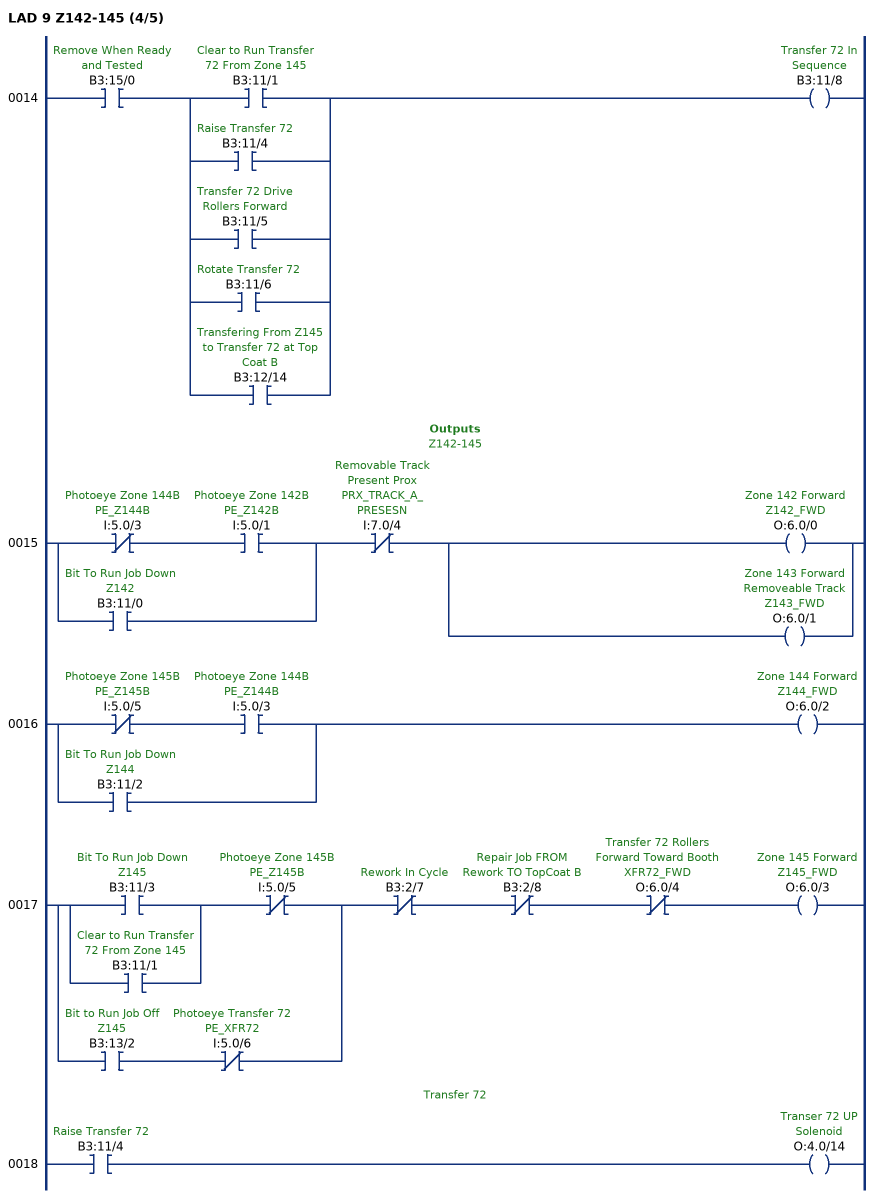
% Rung: 14 %
SOR XIC B3:15/0 BST XIC B3:11/1 NXB XIC B3:11/4 NXB XIC B3:11/5 NXB XIC B3:11/6 NXB XIC B3:12/14 BND OTE B3:11/8 EOR
%   B3:15/0  "Remove When Ready and Tested" %
%   B3:11/1  "Clear to Run Transfer 72 From Zone 145" %
%   B3:11/4  "Raise Transfer 72" %
%   B3:11/5  "Transfer 72 Drive Rollers Forward" %
%   B3:11/6  "Rotate Transfer 72" %
%   B3:12/14  "Transfering From Z145 to Transfer 72 at Top Coat B" %
%   B3:11/8  "Transfer 72 In Sequence" %
% Rung: 15 %
% TITLE: Outputs %
% Z142-145 %
SOR BST XIO I:5.0/3 XIC I:5.0/1 NXB XIC B3:11/0 BND XIO I:7.0/4 BST OTE O:6.0/0 NXB OTE O:6.0/1 BND EOR
%   I:5.0/3  PE_Z144B  "Photoeye Zone 144B" %
%   I:5.0/1  PE_Z142B  "Photoeye Zone 142B" %
%   B3:11/0  "Bit To Run Job Down Z142" %
%   I:7.0/4  PRX_TRACK_A_PRESESN  "Removable Track Present Prox" %
%   O:6.0/0  Z142_FWD  "Zone 142 Forward" %
%   O:6.0/1  Z143_FWD  "Zone 143 Forward Removeable Track" %
% Rung: 16 %
SOR BST XIO I:5.0/5 XIC I:5.0/3 NXB XIC B3:11/2 BND OTE O:6.0/2 EOR
%   I:5.0/5  PE_Z145B  "Photoeye Zone 145B" %
%   I:5.0/3  PE_Z144B  "Photoeye Zone 144B" %
%   B3:11/2  "Bit To Run Job Down Z144" %
%   O:6.0/2  Z144_FWD  "Zone 144 Forward" %
% Rung: 17 %
SOR BST BST XIC B3:11/3 NXB XIC B3:11/1 BND XIO I:5.0/5 NXB XIC B3:13/2 XIO I:5.0/6 BND XIO B3:2/7 XIO B3:2/8 XIO O:6.0/4 OTE O:6.0/3 EOR
%   B3:11/3  "Bit To Run Job Down Z145" %
%   B3:11/1  "Clear to Run Transfer 72 From Zone 145" %
%   I:5.0/5  PE_Z145B  "Photoeye Zone 145B" %
%   B3:13/2  "Bit to Run Job Off Z145" %
%   I:5.0/6  PE_XFR72  "Photoeye Transfer 72" %
%   B3:2/7  "Rework In Cycle" %
%   B3:2/8  "Repair Job FROM Rework TO TopCoat B" %
%   O:6.0/4  XFR72_FWD  "Transfer 72 Rollers Forward Toward Booth" %
%   O:6.0/3  Z145_FWD  "Zone 145 Forward" %
% Rung: 18 %
% Transfer 72 %
SOR XIC B3:11/4 OTE O:4.0/14 EOR
%   B3:11/4  "Raise Transfer 72" %
%   O:4.0/14  "Transer 72 UP Solenoid" %

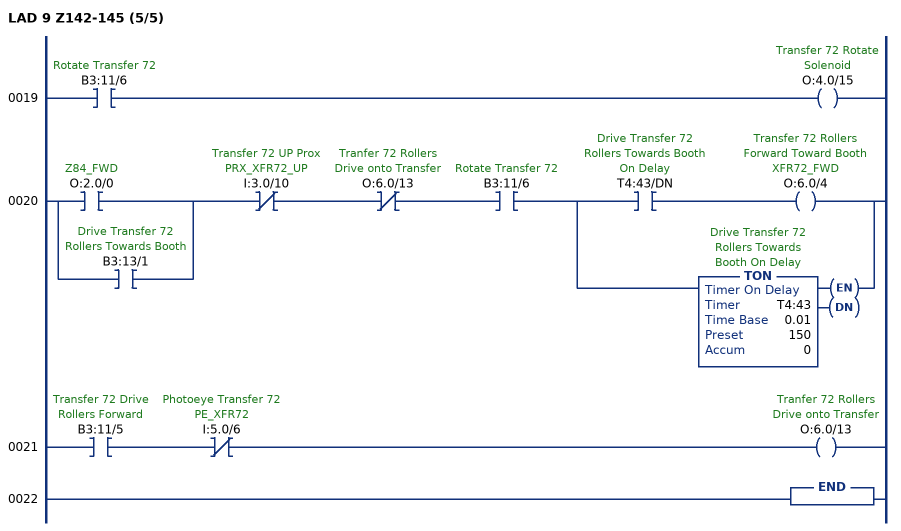
% Rung: 19 %
SOR XIC B3:11/6 OTE O:4.0/15 EOR
%   B3:11/6  "Rotate Transfer 72" %
%   O:4.0/15  "Transfer 72 Rotate Solenoid" %
% Rung: 20 %
SOR BST XIC O:2.0/0 NXB XIC B3:13/1 BND XIO I:3.0/10 XIO O:6.0/13 XIC B3:11/6 BST XIC T4:43/DN OTE O:6.0/4 NXB TON T4:43 0.01 150 0 BND EOR
%   O:2.0/0  Z84_FWD %
%   B3:13/1  "Drive Transfer 72 Rollers Towards Booth" %
%   I:3.0/10  PRX_XFR72_UP  "Transfer 72 UP Prox" %
%   O:6.0/13  "Tranfer 72 Rollers Drive onto Transfer" %
%   B3:11/6  "Rotate Transfer 72" %
%   T4:43  "Drive Transfer 72 Rollers Towards Booth On Delay" %
%   O:6.0/4  XFR72_FWD  "Transfer 72 Rollers Forward Toward Booth" %
% Rung: 21 %
SOR XIC B3:11/5 XIO I:5.0/6 OTE O:6.0/13 EOR
%   B3:11/5  "Transfer 72 Drive Rollers Forward" %
%   I:5.0/6  PE_XFR72  "Photoeye Transfer 72" %
%   O:6.0/13  "Tranfer 72 Rollers Drive onto Transfer" %
% Rung: 22 %
SOR END EOR

LADDER 10 "TO_GLAZE"
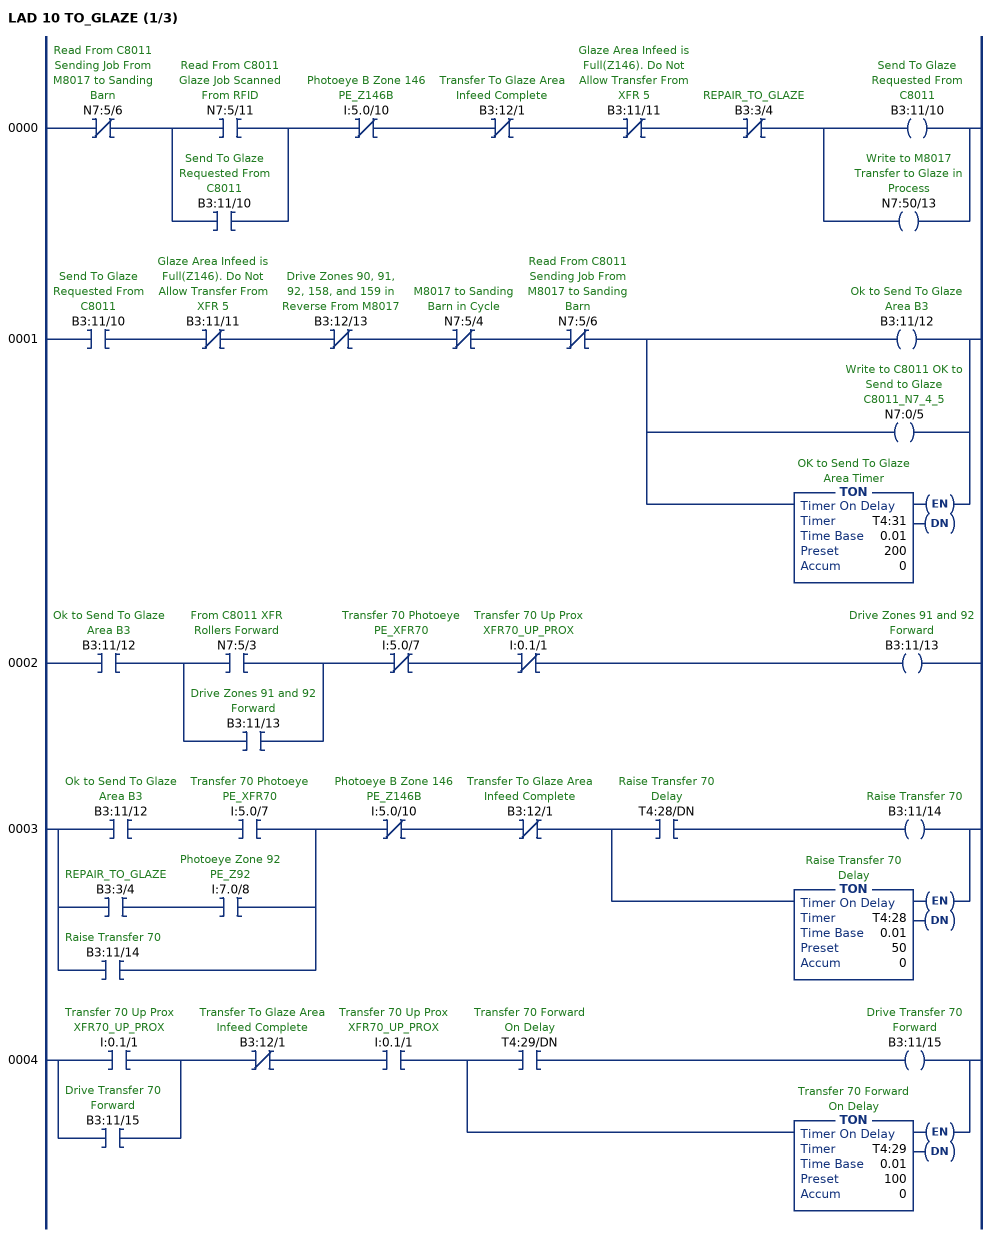
% Rung: 0 %
SOR XIO N7:5/6 BST XIC N7:5/11 NXB XIC B3:11/10 BND XIO I:5.0/10 XIO B3:12/1 XIO B3:11/11 XIO B3:3/4 BST OTE B3:11/10 NXB OTE N7:50/13 BND EOR
%   N7:5/6  "Read From C8011 Sending Job From M8017 to Sanding Barn" %
%   N7:5/11  "Read From C8011 Glaze Job Scanned From RFID" %
%   B3:11/10  "Send To Glaze Requested From C8011" %
%   I:5.0/10  PE_Z146B  "Photoeye B Zone 146" %
%   B3:12/1  "Transfer To Glaze Area Infeed Complete" %
%   B3:11/11  "Glaze Area Infeed is Full(Z146). Do Not Allow Transfer From XFR 5" %
%   B3:3/4  REPAIR_TO_GLAZE %
%   N7:50/13  "Write to M8017 Transfer to Glaze in Process" %
% Rung: 1 %
SOR XIC B3:11/10 XIO B3:11/11 XIO B3:12/13 XIO N7:5/4 XIO N7:5/6 BST BST OTE B3:11/12 NXB OTE N7:0/5 BND NXB TON T4:31 0.01 200 0 BND EOR
%   B3:11/10  "Send To Glaze Requested From C8011" %
%   B3:11/11  "Glaze Area Infeed is Full(Z146). Do Not Allow Transfer From XFR 5" %
%   B3:12/13  "Drive Zones 90, 91, 92, 158, and 159 in Reverse From M8017" %
%   N7:5/4  "M8017 to Sanding Barn in Cycle" %
%   N7:5/6  "Read From C8011 Sending Job From M8017 to Sanding Barn" %
%   B3:11/12  B3  "Ok to Send To Glaze Area" %
%   N7:0/5  C8011_N7_4_5  "Write to C8011 OK to Send to Glaze" %
%   T4:31  "OK to Send To Glaze Area Timer" %
% Rung: 2 %
SOR XIC B3:11/12 BST XIC N7:5/3 NXB XIC B3:11/13 BND XIO I:5.0/7 XIO I:0.1/1 OTE B3:11/13 EOR
%   B3:11/12  B3  "Ok to Send To Glaze Area" %
%   N7:5/3  "From C8011 XFR Rollers Forward" %
%   B3:11/13  "Drive Zones 91 and 92 Forward" %
%   I:5.0/7  PE_XFR70  "Transfer 70 Photoeye" %
%   I:0.1/1  XFR70_UP_PROX  "Transfer 70 Up Prox" %
% Rung: 3 %
SOR BST XIC B3:11/12 XIC I:5.0/7 NXB XIC B3:3/4 XIC I:7.0/8 NXB XIC B3:11/14 BND XIO I:5.0/10 XIO B3:12/1 BST XIC T4:28/DN OTE B3:11/14 NXB TON T4:28 0.01 50 0 BND EOR
%   B3:11/12  B3  "Ok to Send To Glaze Area" %
%   I:5.0/7  PE_XFR70  "Transfer 70 Photoeye" %
%   B3:3/4  REPAIR_TO_GLAZE %
%   I:7.0/8  PE_Z92  "Photoeye Zone 92" %
%   B3:11/14  "Raise Transfer 70" %
%   I:5.0/10  PE_Z146B  "Photoeye B Zone 146" %
%   B3:12/1  "Transfer To Glaze Area Infeed Complete" %
%   T4:28  "Raise Transfer 70 Delay" %
% Rung: 4 %
SOR BST XIC I:0.1/1 NXB XIC B3:11/15 BND XIO B3:12/1 XIC I:0.1/1 BST XIC T4:29/DN OTE B3:11/15 NXB TON T4:29 0.01 100 0 BND EOR
%   I:0.1/1  XFR70_UP_PROX  "Transfer 70 Up Prox" %
%   B3:11/15  "Drive Transfer 70 Forward" %
%   B3:12/1  "Transfer To Glaze Area Infeed Complete" %
%   T4:29  "Transfer 70 Forward On Delay" %

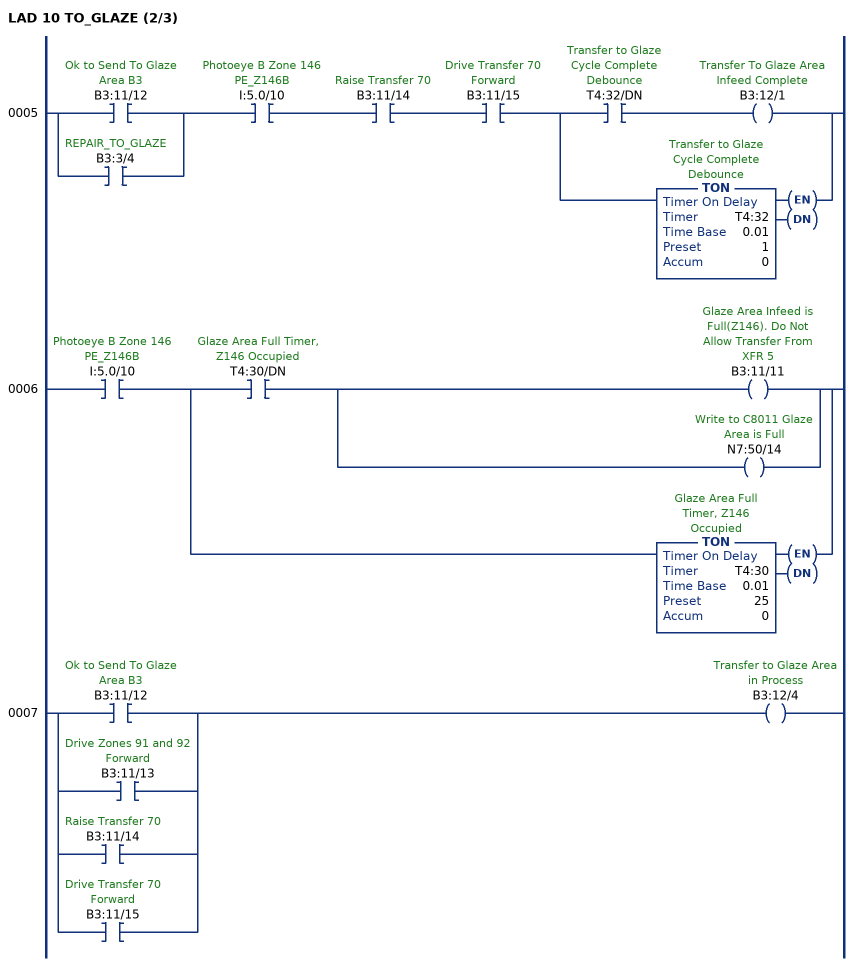
% Rung: 5 %
SOR BST XIC B3:11/12 NXB XIC B3:3/4 BND XIC I:5.0/10 XIC B3:11/14 XIC B3:11/15 BST XIC T4:32/DN OTE B3:12/1 NXB TON T4:32 0.01 1 0 BND EOR
%   B3:11/12  B3  "Ok to Send To Glaze Area" %
%   B3:3/4  REPAIR_TO_GLAZE %
%   I:5.0/10  PE_Z146B  "Photoeye B Zone 146" %
%   B3:11/14  "Raise Transfer 70" %
%   B3:11/15  "Drive Transfer 70 Forward" %
%   T4:32  "Transfer to Glaze Cycle Complete Debounce" %
%   B3:12/1  "Transfer To Glaze Area Infeed Complete" %
% Rung: 6 %
SOR XIC I:5.0/10 BST XIC T4:30/DN BST OTE B3:11/11 NXB OTE N7:50/14 BND NXB TON T4:30 0.01 25 0 BND EOR
%   I:5.0/10  PE_Z146B  "Photoeye B Zone 146" %
%   T4:30  "Glaze Area Full Timer, Z146 Occupied" %
%   B3:11/11  "Glaze Area Infeed is Full(Z146). Do Not Allow Transfer From XFR 5" %
%   N7:50/14  "Write to C8011 Glaze Area is Full" %
% Rung: 7 %
SOR BST XIC B3:11/12 NXB XIC B3:11/13 NXB XIC B3:11/14 NXB XIC B3:11/15 BND OTE B3:12/4 EOR
%   B3:11/12  B3  "Ok to Send To Glaze Area" %
%   B3:11/13  "Drive Zones 91 and 92 Forward" %
%   B3:11/14  "Raise Transfer 70" %
%   B3:11/15  "Drive Transfer 70 Forward" %
%   B3:12/4  "Transfer to Glaze Area in Process" %

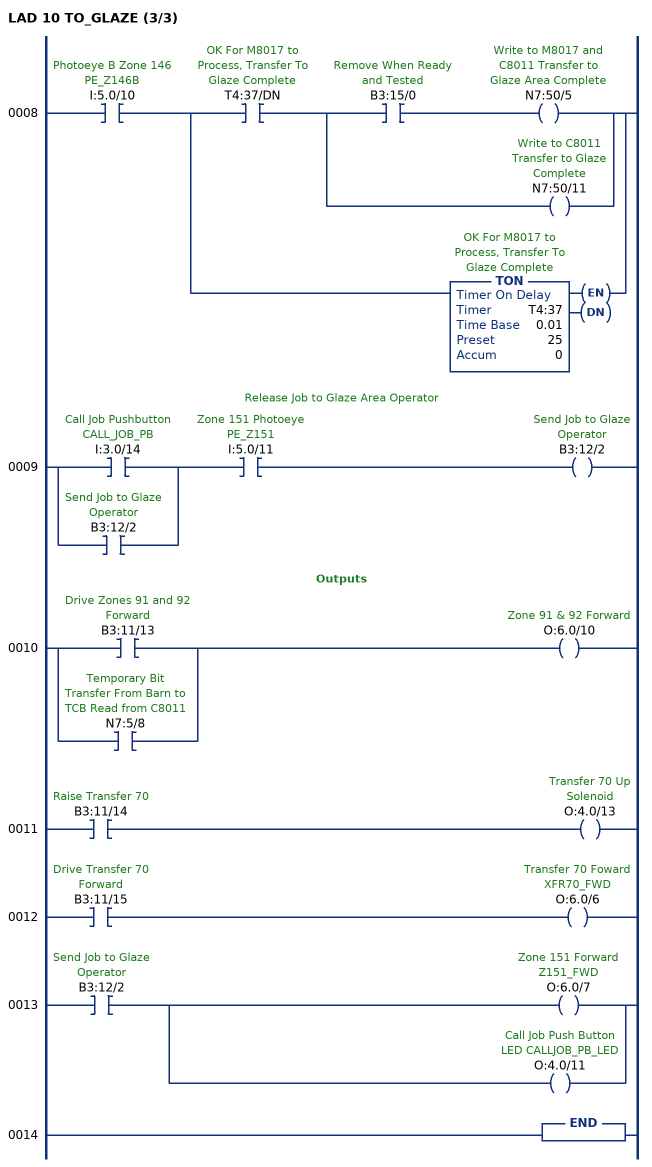
% Rung: 8 %
SOR XIC I:5.0/10 BST XIC T4:37/DN BST XIC B3:15/0 OTE N7:50/5 NXB OTE N7:50/11 BND NXB TON T4:37 0.01 25 0 BND EOR
%   I:5.0/10  PE_Z146B  "Photoeye B Zone 146" %
%   T4:37  "OK For M8017 to Process, Transfer To Glaze Complete" %
%   B3:15/0  "Remove When Ready and Tested" %
%   N7:50/5  "Write to M8017 and C8011 Transfer to Glaze Area Complete" %
%   N7:50/11  "Write to C8011 Transfer to Glaze Complete" %
% Rung: 9 %
% Release Job to Glaze Area Operator %
SOR BST XIC I:3.0/14 NXB XIC B3:12/2 BND XIC I:5.0/11 OTE B3:12/2 EOR
%   I:3.0/14  CALL_JOB_PB  "Call Job Pushbutton" %
%   B3:12/2  "Send Job to Glaze Operator" %
%   I:5.0/11  PE_Z151  "Zone 151 Photoeye" %
% Rung: 10 %
% TITLE: Outputs %
SOR BST XIC B3:11/13 NXB XIC N7:5/8 BND OTE O:6.0/10 EOR
%   B3:11/13  "Drive Zones 91 and 92 Forward" %
%   N7:5/8  "Temporary Bit Transfer From Barn to TCB Read from C8011" %
%   O:6.0/10  "Zone 91 & 92 Forward" %
% Rung: 11 %
SOR XIC B3:11/14 OTE O:4.0/13 EOR
%   B3:11/14  "Raise Transfer 70" %
%   O:4.0/13  "Transfer 70 Up Solenoid" %
% Rung: 12 %
SOR XIC B3:11/15 OTE O:6.0/6 EOR
%   B3:11/15  "Drive Transfer 70 Forward" %
%   O:6.0/6  XFR70_FWD  "Transfer 70 Foward" %
% Rung: 13 %
SOR XIC B3:12/2 BST OTE O:6.0/7 NXB OTE O:4.0/11 BND EOR
%   B3:12/2  "Send Job to Glaze Operator" %
%   O:6.0/7  Z151_FWD  "Zone 151 Forward" %
%   O:4.0/11  CALLJOB_PB_LED  "Call Job Push Button LED" %
% Rung: 14 %
SOR END EOR

LADDER 11 "FROM_GLAZE"
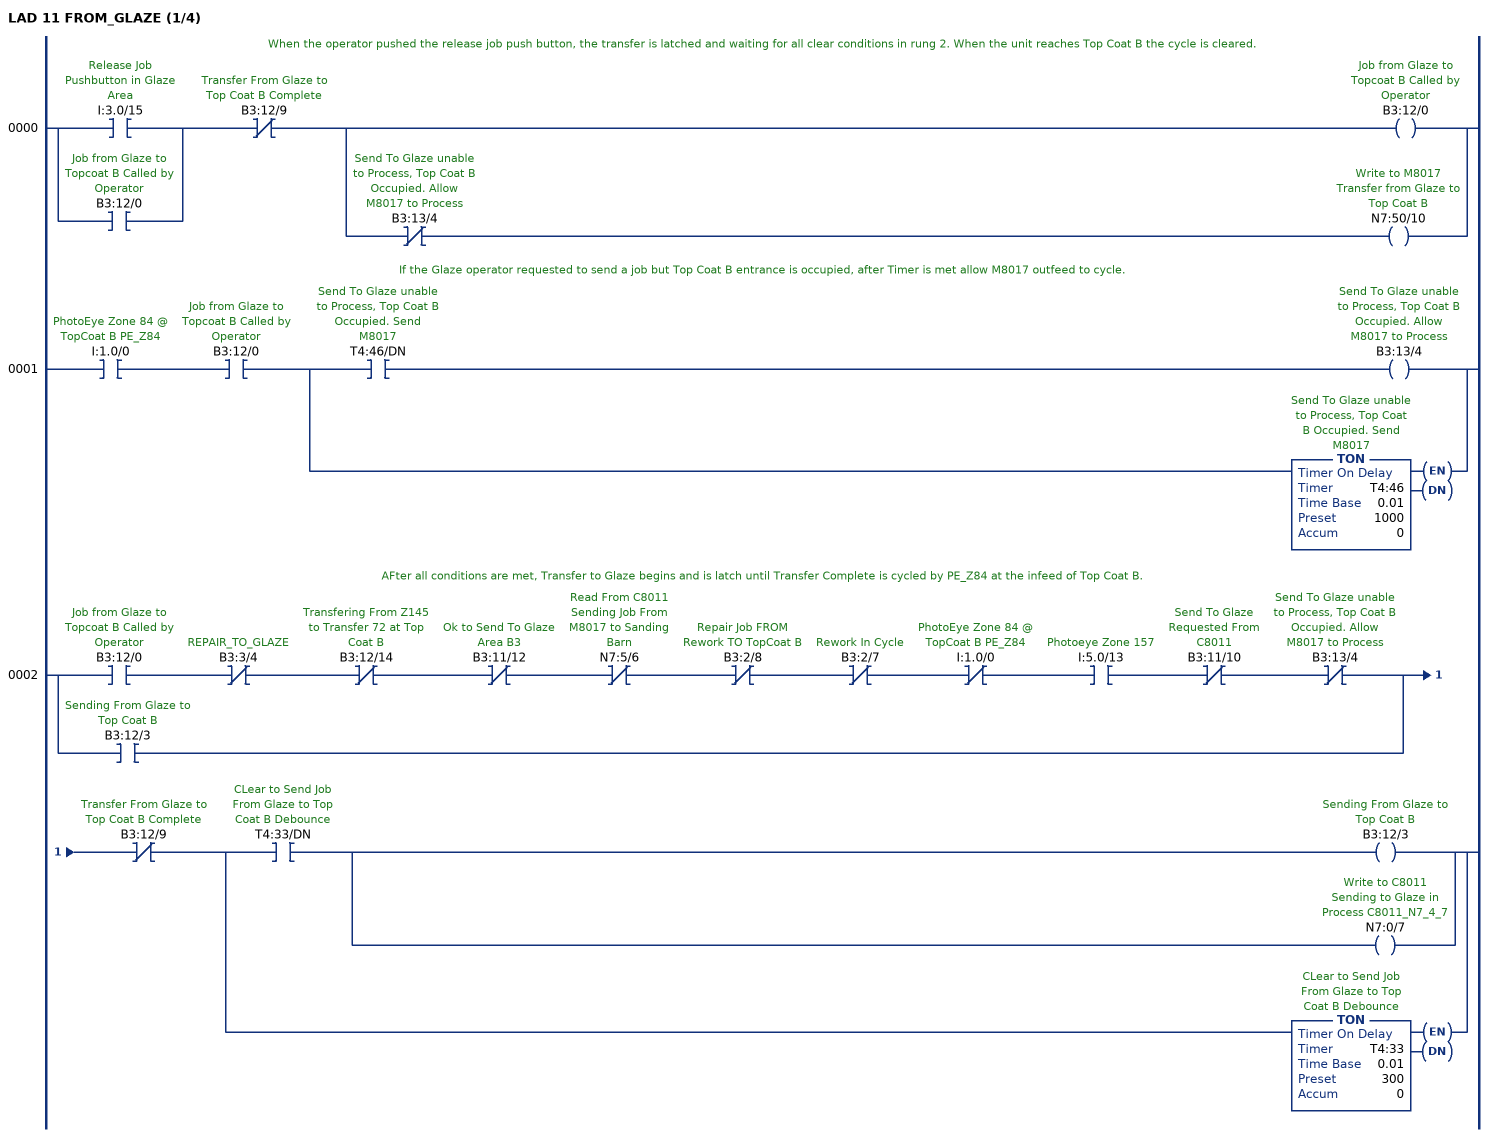
% Rung: 0 %
% When the operator pushed the release job push button, the transfer is latched and waiting for all clear conditions in rung 2. When the unit reaches Top Coat B the cycle is cleared. %
SOR BST XIC I:3.0/15 NXB XIC B3:12/0 BND XIO B3:12/9 BST OTE B3:12/0 NXB XIO B3:13/4 OTE N7:50/10 BND EOR
%   I:3.0/15  "Release Job Pushbutton in Glaze Area" %
%   B3:12/0  "Job from Glaze to Topcoat B Called by Operator" %
%   B3:12/9  "Transfer From Glaze to Top Coat B Complete" %
%   B3:13/4  "Send To Glaze unable to Process, Top Coat B Occupied. Allow M8017 to Process" %
%   N7:50/10  "Write to M8017 Transfer from Glaze to Top Coat B" %
% Rung: 1 %
% If the Glaze operator requested to send a job but Top Coat B entrance is occupied, after Timer is met allow M8017 outfeed to cycle. %
SOR XIC I:1.0/0 XIC B3:12/0 BST XIC T4:46/DN OTE B3:13/4 NXB TON T4:46 0.01 1000 0 BND EOR
%   I:1.0/0  PE_Z84  "PhotoEye Zone 84 @ TopCoat B" %
%   B3:12/0  "Job from Glaze to Topcoat B Called by Operator" %
%   T4:46  "Send To Glaze unable to Process, Top Coat B Occupied. Send M8017" %
%   B3:13/4  "Send To Glaze unable to Process, Top Coat B Occupied. Allow M8017 to Process" %
% Rung: 2 %
% AFter all conditions are met, Transfer to Glaze begins and is latch until Transfer Complete is cycled by PE_Z84 at the infeed of Top Coat B. %
SOR BST XIC B3:12/0 XIO B3:3/4 XIO B3:12/14 XIO B3:11/12 XIO N7:5/6 XIO B3:2/8 XIO B3:2/7 XIO I:1.0/0 XIC I:5.0/13 XIO B3:11/10 XIO B3:13/4 NXB XIC B3:12/3 BND XIO B3:12/9 BST XIC T4:33/DN BST OTE B3:12/3 NXB OTE N7:0/7 BND NXB TON T4:33 0.01 300 0 BND EOR
%   B3:12/0  "Job from Glaze to Topcoat B Called by Operator" %
%   B3:3/4  REPAIR_TO_GLAZE %
%   B3:12/14  "Transfering From Z145 to Transfer 72 at Top Coat B" %
%   B3:11/12  B3  "Ok to Send To Glaze Area" %
%   N7:5/6  "Read From C8011 Sending Job From M8017 to Sanding Barn" %
%   B3:2/8  "Repair Job FROM Rework TO TopCoat B" %
%   B3:2/7  "Rework In Cycle" %
%   I:1.0/0  PE_Z84  "PhotoEye Zone 84 @ TopCoat B" %
%   I:5.0/13  "Photoeye Zone 157" %
%   B3:11/10  "Send To Glaze Requested From C8011" %
%   B3:13/4  "Send To Glaze unable to Process, Top Coat B Occupied. Allow M8017 to Process" %
%   B3:12/3  "Sending From Glaze to Top Coat B" %
%   B3:12/9  "Transfer From Glaze to Top Coat B Complete" %
%   T4:33  "CLear to Send Job From Glaze to Top Coat B Debounce" %
%   N7:0/7  C8011_N7_4_7  "Write to C8011 Sending to Glaze in Process" %

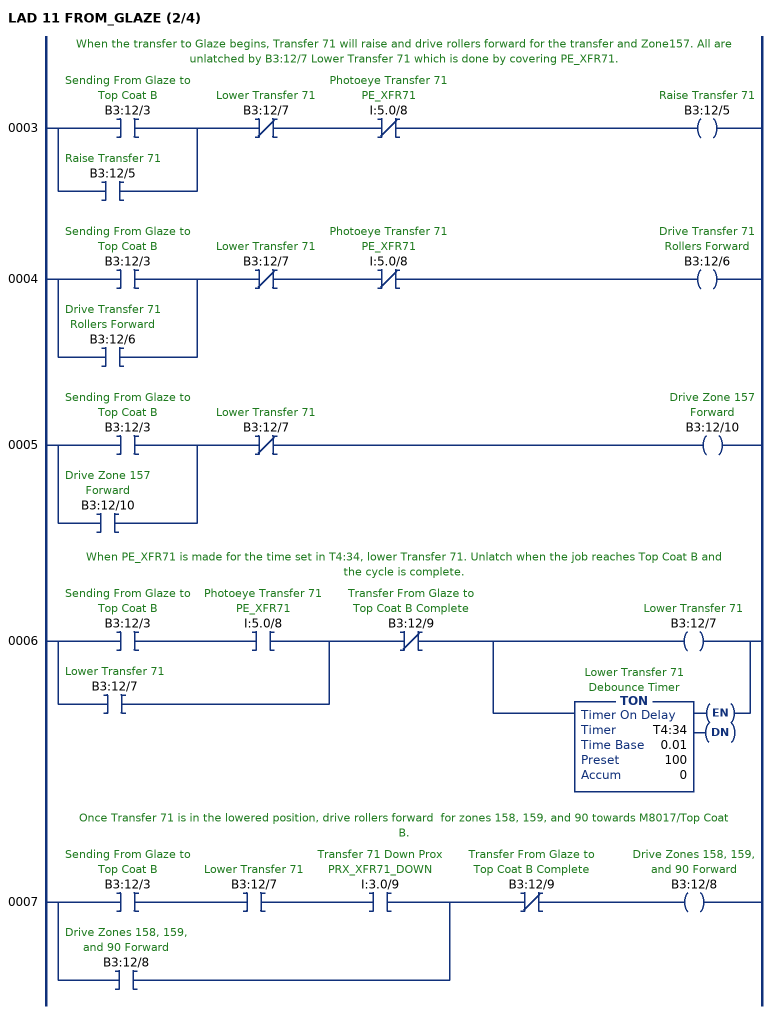
% Rung: 3 %
% When the transfer to Glaze begins, Transfer 71 will raise and drive rollers forward for the transfer and Zone157. All are unlatched by B3:12/7 Lower Transfer 71 which is done by covering PE_XFR71. %
SOR BST XIC B3:12/3 NXB XIC B3:12/5 BND XIO B3:12/7 XIO I:5.0/8 OTE B3:12/5 EOR
%   B3:12/3  "Sending From Glaze to Top Coat B" %
%   B3:12/5  "Raise Transfer 71" %
%   B3:12/7  "Lower Transfer 71" %
%   I:5.0/8  PE_XFR71  "Photoeye Transfer 71" %
% Rung: 4 %
SOR BST XIC B3:12/3 NXB XIC B3:12/6 BND XIO B3:12/7 XIO I:5.0/8 OTE B3:12/6 EOR
%   B3:12/3  "Sending From Glaze to Top Coat B" %
%   B3:12/6  "Drive Transfer 71 Rollers Forward" %
%   B3:12/7  "Lower Transfer 71" %
%   I:5.0/8  PE_XFR71  "Photoeye Transfer 71" %
% Rung: 5 %
SOR BST XIC B3:12/3 NXB XIC B3:12/10 BND XIO B3:12/7 OTE B3:12/10 EOR
%   B3:12/3  "Sending From Glaze to Top Coat B" %
%   B3:12/10  "Drive Zone 157 Forward" %
%   B3:12/7  "Lower Transfer 71" %
% Rung: 6 %
% When PE_XFR71 is made for the time set in T4:34, lower Transfer 71. Unlatch when the job reaches Top Coat B and the cycle is complete. %
SOR BST XIC B3:12/3 XIC I:5.0/8 NXB XIC B3:12/7 BND XIO B3:12/9 BST OTE B3:12/7 NXB TON T4:34 0.01 100 0 BND EOR
%   B3:12/3  "Sending From Glaze to Top Coat B" %
%   I:5.0/8  PE_XFR71  "Photoeye Transfer 71" %
%   B3:12/7  "Lower Transfer 71" %
%   B3:12/9  "Transfer From Glaze to Top Coat B Complete" %
%   T4:34  "Lower Transfer 71 Debounce Timer" %
% Rung: 7 %
% Once Transfer 71 is in the lowered position, drive rollers forward  for zones 158, 159, and 90 towards M8017/Top Coat B. %
SOR BST XIC B3:12/3 XIC B3:12/7 XIC I:3.0/9 NXB XIC B3:12/8 BND XIO B3:12/9 OTE B3:12/8 EOR
%   B3:12/3  "Sending From Glaze to Top Coat B" %
%   B3:12/7  "Lower Transfer 71" %
%   I:3.0/9  PRX_XFR71_DOWN  "Transfer 71 Down Prox" %
%   B3:12/8  "Drive Zones 158, 159, and 90 Forward" %
%   B3:12/9  "Transfer From Glaze to Top Coat B Complete" %

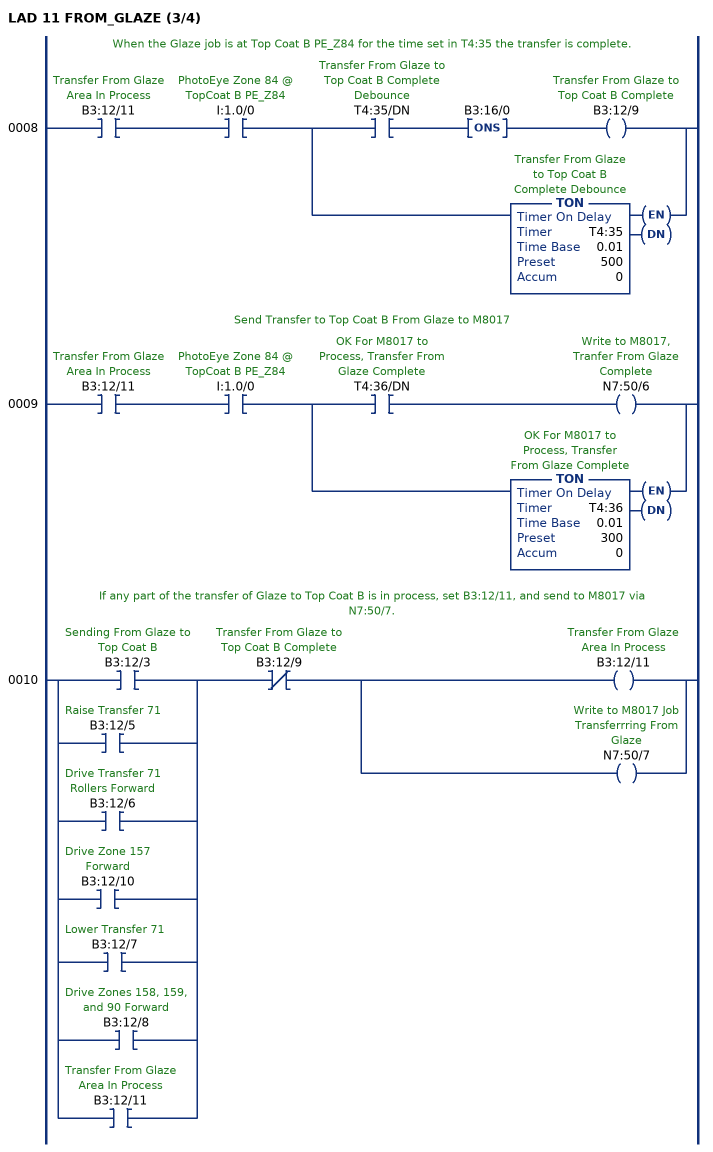
% Rung: 8 %
% When the Glaze job is at Top Coat B PE_Z84 for the time set in T4:35 the transfer is complete. %
SOR XIC B3:12/11 XIC I:1.0/0 BST XIC T4:35/DN ONS B3:16/0 OTE B3:12/9 NXB TON T4:35 0.01 500 0 BND EOR
%   B3:12/11  "Transfer From Glaze Area In Process" %
%   I:1.0/0  PE_Z84  "PhotoEye Zone 84 @ TopCoat B" %
%   T4:35  "Transfer From Glaze to Top Coat B Complete Debounce" %
%   B3:12/9  "Transfer From Glaze to Top Coat B Complete" %
% Rung: 9 %
% Send Transfer to Top Coat B From Glaze to M8017 %
SOR XIC B3:12/11 XIC I:1.0/0 BST XIC T4:36/DN OTE N7:50/6 NXB TON T4:36 0.01 300 0 BND EOR
%   B3:12/11  "Transfer From Glaze Area In Process" %
%   I:1.0/0  PE_Z84  "PhotoEye Zone 84 @ TopCoat B" %
%   T4:36  "OK For M8017 to Process, Transfer From Glaze Complete" %
%   N7:50/6  "Write to M8017, Tranfer From Glaze Complete" %
% Rung: 10 %
% If any part of the transfer of Glaze to Top Coat B is in process, set B3:12/11, and send to M8017 via N7:50/7. %
SOR BST XIC B3:12/3 NXB XIC B3:12/5 NXB XIC B3:12/6 NXB XIC B3:12/10 NXB XIC B3:12/7 NXB XIC B3:12/8 NXB XIC B3:12/11 BND XIO B3:12/9 BST OTE B3:12/11 NXB OTE N7:50/7 BND EOR
%   B3:12/3  "Sending From Glaze to Top Coat B" %
%   B3:12/5  "Raise Transfer 71" %
%   B3:12/6  "Drive Transfer 71 Rollers Forward" %
%   B3:12/10  "Drive Zone 157 Forward" %
%   B3:12/7  "Lower Transfer 71" %
%   B3:12/8  "Drive Zones 158, 159, and 90 Forward" %
%   B3:12/11  "Transfer From Glaze Area In Process" %
%   B3:12/9  "Transfer From Glaze to Top Coat B Complete" %
%   N7:50/7  "Write to M8017 Job Transferrring From Glaze" %

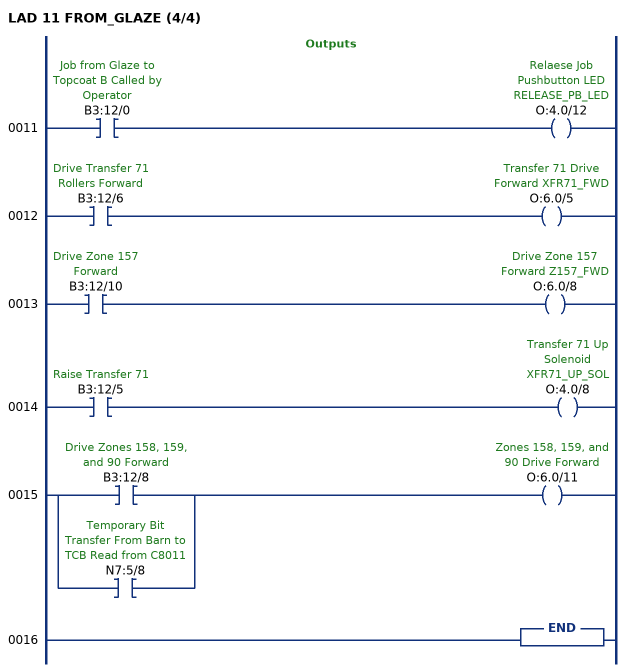
% Rung: 11 %
% TITLE: Outputs %
SOR XIC B3:12/0 OTE O:4.0/12 EOR
%   B3:12/0  "Job from Glaze to Topcoat B Called by Operator" %
%   O:4.0/12  RELEASE_PB_LED  "Relaese Job Pushbutton LED" %
% Rung: 12 %
SOR XIC B3:12/6 OTE O:6.0/5 EOR
%   B3:12/6  "Drive Transfer 71 Rollers Forward" %
%   O:6.0/5  XFR71_FWD  "Transfer 71 Drive Forward" %
% Rung: 13 %
SOR XIC B3:12/10 OTE O:6.0/8 EOR
%   B3:12/10  "Drive Zone 157 Forward" %
%   O:6.0/8  Z157_FWD  "Drive Zone 157 Forward" %
% Rung: 14 %
SOR XIC B3:12/5 OTE O:4.0/8 EOR
%   B3:12/5  "Raise Transfer 71" %
%   O:4.0/8  XFR71_UP_SOL  "Transfer 71 Up Solenoid" %
% Rung: 15 %
SOR BST XIC B3:12/8 NXB XIC N7:5/8 BND OTE O:6.0/11 EOR
%   B3:12/8  "Drive Zones 158, 159, and 90 Forward" %
%   N7:5/8  "Temporary Bit Transfer From Barn to TCB Read from C8011" %
%   O:6.0/11  "Zones 158, 159, and 90 Drive Forward" %
% Rung: 16 %
SOR END EOR

LADDER 12 "TO_BARN"
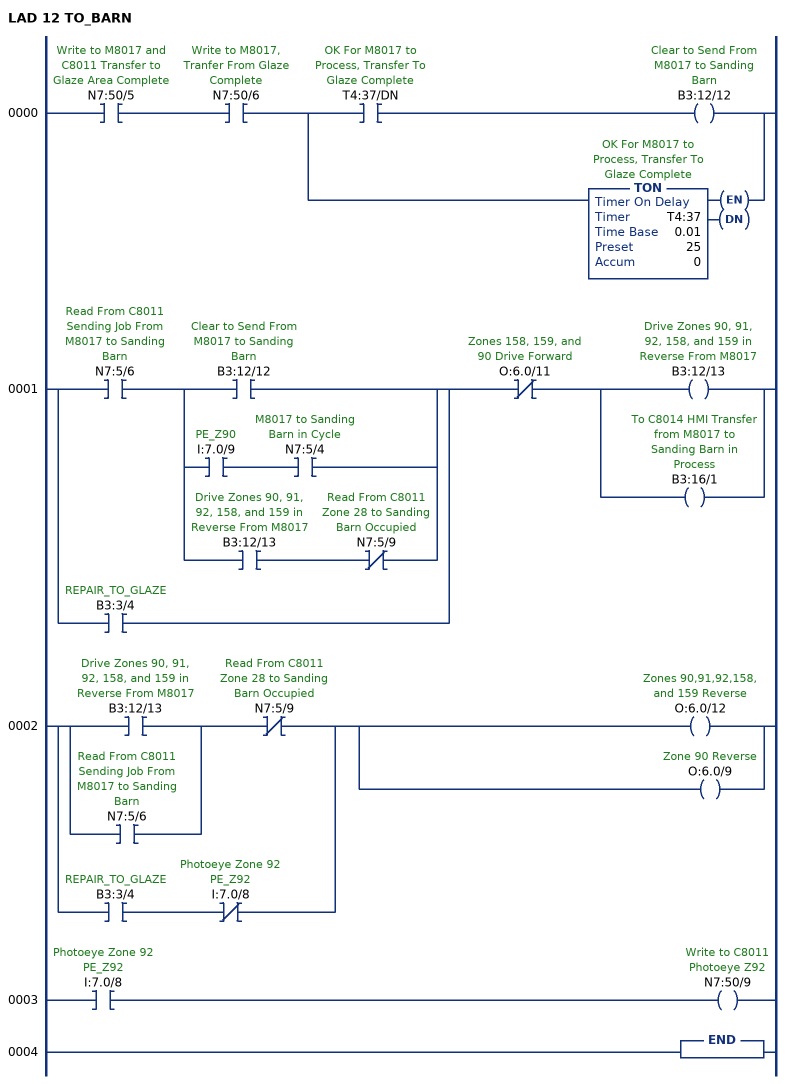
% Rung: 0 %
SOR XIC N7:50/5 XIC N7:50/6 BST XIC T4:37/DN OTE B3:12/12 NXB TON T4:37 0.01 25 0 BND EOR
%   N7:50/5  "Write to M8017 and C8011 Transfer to Glaze Area Complete" %
%   N7:50/6  "Write to M8017, Tranfer From Glaze Complete" %
%   T4:37  "OK For M8017 to Process, Transfer To Glaze Complete" %
%   B3:12/12  "Clear to Send From M8017 to Sanding Barn" %
% Rung: 1 %
SOR BST XIC N7:5/6 BST XIC B3:12/12 NXB XIC I:7.0/9 XIC N7:5/4 NXB XIC B3:12/13 XIO N7:5/9 BND NXB XIC B3:3/4 BND XIO O:6.0/11 BST OTE B3:12/13 NXB OTE B3:16/1 BND EOR
%   N7:5/6  "Read From C8011 Sending Job From M8017 to Sanding Barn" %
%   B3:12/12  "Clear to Send From M8017 to Sanding Barn" %
%   I:7.0/9  PE_Z90 %
%   N7:5/4  "M8017 to Sanding Barn in Cycle" %
%   B3:12/13  "Drive Zones 90, 91, 92, 158, and 159 in Reverse From M8017" %
%   N7:5/9  "Read From C8011 Zone 28 to Sanding Barn Occupied" %
%   B3:3/4  REPAIR_TO_GLAZE %
%   O:6.0/11  "Zones 158, 159, and 90 Drive Forward" %
%   B3:16/1  "To C8014 HMI Transfer from M8017 to Sanding Barn in Process" %
% Rung: 2 %
SOR BST BST XIC B3:12/13 NXB XIC N7:5/6 BND XIO N7:5/9 NXB XIC B3:3/4 XIO I:7.0/8 BND BST OTE O:6.0/12 NXB OTE O:6.0/9 BND EOR
%   B3:12/13  "Drive Zones 90, 91, 92, 158, and 159 in Reverse From M8017" %
%   N7:5/6  "Read From C8011 Sending Job From M8017 to Sanding Barn" %
%   N7:5/9  "Read From C8011 Zone 28 to Sanding Barn Occupied" %
%   B3:3/4  REPAIR_TO_GLAZE %
%   I:7.0/8  PE_Z92  "Photoeye Zone 92" %
%   O:6.0/12  "Zones 90,91,92,158, and 159 Reverse" %
%   O:6.0/9  "Zone 90 Reverse" %
% Rung: 3 %
SOR XIC I:7.0/8 OTE N7:50/9 EOR
%   I:7.0/8  PE_Z92  "Photoeye Zone 92" %
%   N7:50/9  "Write to C8011 Photoeye Z92" %
% Rung: 4 %
SOR END EOR

LADDER 13 "FRM_REPAIR"
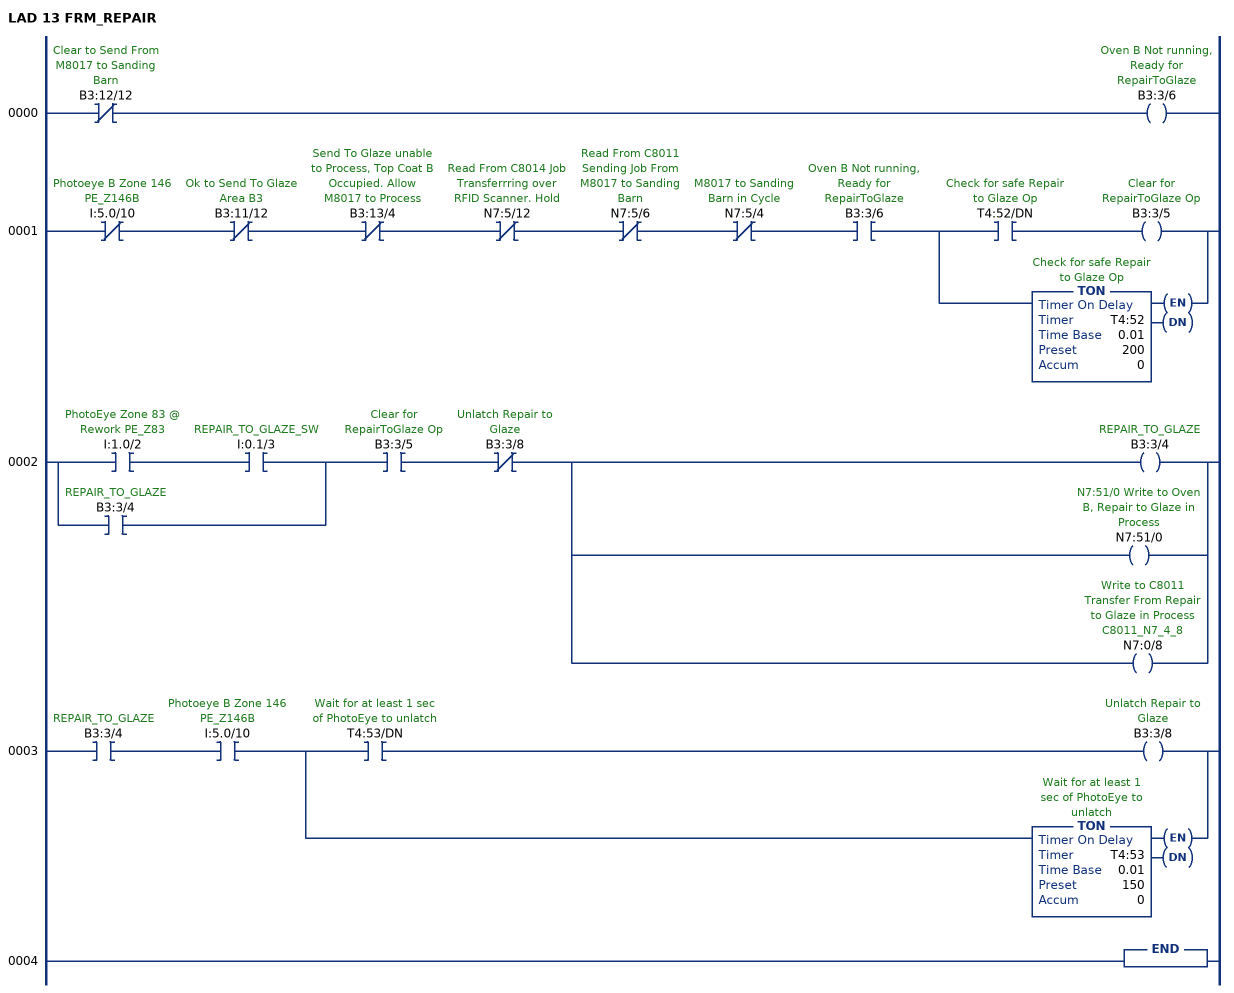
% Rung: 0 %
SOR XIO B3:12/12 OTE B3:3/6 EOR
%   B3:12/12  "Clear to Send From M8017 to Sanding Barn" %
%   B3:3/6  "Oven B Not running, Ready for RepairToGlaze" %
% Rung: 1 %
SOR XIO I:5.0/10 XIO B3:11/12 XIO B3:13/4 XIO N7:5/12 XIO N7:5/6 XIO N7:5/4 XIC B3:3/6 BST XIC T4:52/DN OTE B3:3/5 NXB TON T4:52 0.01 200 0 BND EOR
%   I:5.0/10  PE_Z146B  "Photoeye B Zone 146" %
%   B3:11/12  B3  "Ok to Send To Glaze Area" %
%   B3:13/4  "Send To Glaze unable to Process, Top Coat B Occupied. Allow M8017 to Process" %
%   N7:5/12  "Read From C8014 Job Transferrring over RFID Scanner. Hold" %
%   N7:5/6  "Read From C8011 Sending Job From M8017 to Sanding Barn" %
%   N7:5/4  "M8017 to Sanding Barn in Cycle" %
%   B3:3/6  "Oven B Not running, Ready for RepairToGlaze" %
%   T4:52  "Check for safe Repair to Glaze Op" %
%   B3:3/5  "Clear for RepairToGlaze Op" %
% Rung: 2 %
SOR BST XIC I:1.0/2 XIC I:0.1/3 NXB XIC B3:3/4 BND XIC B3:3/5 XIO B3:3/8 BST OTE B3:3/4 NXB OTE N7:51/0 NXB OTE N7:0/8 BND EOR
%   I:1.0/2  PE_Z83  "PhotoEye Zone 83 @ Rework" %
%   I:0.1/3  REPAIR_TO_GLAZE_SW %
%   B3:3/4  REPAIR_TO_GLAZE %
%   B3:3/5  "Clear for RepairToGlaze Op" %
%   B3:3/8  "Unlatch Repair to Glaze" %
%   N7:51/0  "N7:51/0 Write to Oven B, Repair to Glaze in Process" %
%   N7:0/8  C8011_N7_4_8  "Write to C8011 Transfer From Repair to Glaze in Process" %
% Rung: 3 %
SOR XIC B3:3/4 XIC I:5.0/10 BST XIC T4:53/DN OTE B3:3/8 NXB TON T4:53 0.01 150 0 BND EOR
%   B3:3/4  REPAIR_TO_GLAZE %
%   I:5.0/10  PE_Z146B  "Photoeye B Zone 146" %
%   T4:53  "Wait for at least 1 sec of PhotoEye to unlatch" %
%   B3:3/8  "Unlatch Repair to Glaze" %
% Rung: 4 %
SOR END EOR

OTHER DOCUMENTED ADDRESSES
  B3:3/7  "XFR70 To Glaze from Repair"
  B3:4/0  SEQ_POL_0  "Sequence Polish Job at ZPOL_1 Ready"
  B3:4/1  SEQ_POL_1  "Sequence Polish Clear ZPOL_7"
  B3:4/2  SEQ_POL_2  "Sequence Polish Job at Transfer 1 End of Belt"
  B3:4/3  SEQ_POL_3  "Sequence Polish Job at Zone Transfer 1 Ready"
  B3:4/4  SEQ_POL_4  "Sequence Polish Job Clear ZX1"
  B10:4/1  IPB_POL_EN  "Interface PushButton Enable Polish"
  I:0.0/0  MCR_OK
  I:0.0/6  PR_XFR11_DN
  I:0.0/7  PE_A
  I:0.0/10  PE_Z89A
  I:0.0/11  PR_XFR12_UP
  I:0.0/15  PR_XFR13_DN
  I:0.1/2  PRX_XFR70_DOWN  "Transfer 70 Down Prox"
  I:1.0/3  PE_Z86
  I:1.0/6  PE_Z87
  I:1.0/7  PE_Z88
  I:3.0/13  PRX_XFR72_90  "Transfer 72 90 Degree Prox"
  I:5.0/0  PE_Z142A  "Photoeye Start Zone 142A"
  I:5.0/2  PE_Z144A  "Photoeye Start Zone 144A"
  I:5.0/4  PE_Z145A  "Photoeye Start Zone 145A"
  I:7.0/0  PR_XFR8_DR
  I:7.0/1  PR_XFR8_HM
  I:7.0/2  PR_XFR8_90
  I:7.0/3  PR_M8011_DR_OP
  I:7.0/5  PR_XFR9_DN
  I:7.0/6  PR_XFR9_DR
  I:7.0/7  PR_XFR9_HM
  I:7.0/10  PE_Z55A
  I:7.0/11  PR_XFR10_UP
  I:7.0/12  PR_XFR10_DN
  MG19:11/3  "Write N7:51 TO M8017"
  N7:1/1  "From C8011 XFR 69 Forward"
  N7:1/5  C8011_N7_5_5  "Writing FROM C8011 Toggle TopCoat B Mode 1 = TopCoat B 0 = Sanding Barn"
  N7:1/6  "From C8011 Sending Job to Sanding Barn"
  N7:5/2  "SEND REWORK FROM TOPCOAT A"
  N7:5/7  "Temporary Bit Transfer From Barn to TCB Read from C8011"
  N7:10/0  "READ FROM M8017 N7:0 InFeed In Cycle TO N7:10/0"
  N7:50/8  "Write to C8011 Glaze Area is Full"
  N7:70  "Glaze Outfeed to Top Coat B Step"
  O:0.0/0  MCR_LED
  O:2.0/10  Z70_FWD
  O:3.0/8  "Gate Actuator - Close"
  O:3.0/9  "Gate Actuator - Open"
  O:4.0/6  XFR72_UP_SOLENOID  "Transer 72 UP Solenoid"
  O:4.0/7  XFR72_ROT_SOLENOID  "Transfer 72 Rotate Solenoid"
  O:5.0/0  Z54_FWD
  O:5.0/1  Z55_FWD
  O:5.0/2  XFR10_FWD
  O:5.0/3  Z57_FWD
  PE_Z51A  
  T4:22  "Delay RFID Match AND Job @ Rework AND NOT From Rework, To TopCoat B"
  T4:47  "Repair to Glaze, Send request"
  T4:69  "Repair Job in Que to go to Top Coat B. Hold Z145"

COMMENTS NOT ATTACHED TO A CURRENT RUNG
  O:0.0/11: If no humans or robots are at the gate and the gate is not fully closed, illuminate the two "Close" buttons. If the gate is actively closing, the light with flash.
  O:3.0/8: The gate will begin to open when the following conditions are met simultaneously:
    1. A human and/or robot has requested access to the gate area.
    2. The gate is not currently open.
    3. No job is actively transferring over the gate.
    
    The gate opener will shut off when the "Gate Open" proximity switch is triggered.
  O:0.0/10: If a human or a robot is at the gate and the gate is not fully open, illuminate the two "Open" buttons. If the gate is actively opening, the light will flash.
  O:3.0/9: If the gate is open and has no humans or robots requesting access, close the gate.
  B3:8/1: When the robot signals that it is finished travelling through the gate, the program will unmark that the gate area has a robot user.
  B3:11/10: From C8011 to Glazing Area

DATA TABLE (non-zero values as saved)
DATA B3
% B3:0 % 0X4C34 0X0027 0X5A52 0X0000 0X0000 0X0080 0X0001 0X0000 0X0000 0X0000
% B3:10 % 0X2000 0X0000 0X0000 0X0001 0X0001 0X0000 0X0000 0X0000 0X0000 0X0000
DATA T4
% .PRE .ACC %
% T4:0 % 1000 0
% T4:1 % 1 0
% T4:2 % 1 1
% T4:3 % 100 0
% T4:4 % 400 0
% T4:5 % 800 800
% T4:6 % 500 500
% T4:7 % 100 0
% T4:8 % 600 321
% T4:9 % 500 0
% T4:10 % 120 0
% T4:11 % 200 200
% T4:12 % 200 200
% T4:13 % 500 0
% T4:14 % 500 0
% T4:15 % 3000 0
% T4:16 % 105 0
% T4:17 % 1200 1200
% T4:18 % 100 0
% T4:19 % 10 0
% T4:20 % 500 0
% T4:21 % 10 1
% T4:22 % 50 0
% T4:23 % 100 100
% T4:24 % 15 0
% T4:25 % 50 0
% T4:26 % 50 0
% T4:27 % 500 0
% T4:28 % 50 0
% T4:29 % 100 0
% T4:30 % 25 0
% T4:31 % 200 0
% T4:32 % 1 0
% T4:33 % 300 0
% T4:34 % 100 0
% T4:35 % 500 0
% T4:36 % 300 0
% T4:37 % 25 0
% T4:38 % 200 0
% T4:39 % 500 0
% T4:40 % 300 0
% T4:41 % 50 0
% T4:42 % 300 300
% T4:43 % 150 0
% T4:44 % 400 0
% T4:45 % 250 0
% T4:46 % 1000 0
% T4:47 % 500 0
% T4:49 % 1000 0
% T4:50 % 8 0
% T4:51 % 30 0
% T4:52 % 200 0
% T4:53 % 150 0
DATA C5
% .PRE .ACC %
% C5:0 % 1 1
% C5:1 % 1 0
DATA N7
% N7:0 % 0 -31728 0 0 0 -32752 0 0 0 0
% N7:50 % 8 0 0 0 0 0 0 0 0 0
% N7:60 % 3 0 0 0 0 0 0 0 0 0
% N7:90 % 46 0 0 0 0 0 0 0 0 0
DATA ST9
% ST9:2 % "!"
% ST9:3 % "71086036"
% ST9:4 % "71085766"
% ST9:5 % "71085999"
% ST9:6 % "71086004"
% ST9:7 % "71086000"
% ST9:8 % "71086001"
% ST9:9 % "71085720"
% ST9:10 % "71086002"
% ST9:11 % "71086003"
% ST9:12 % "71086040"
% ST9:13 % "71086039"
% ST9:14 % "71086038"
% ST9:15 % "71086041"
% ST9:16 % "71086033"
% ST9:17 % "71086035"
% ST9:18 % "71085765"
% ST9:19 % "71086037"
% ST9:20 % "71085766"
